PROGRAM MAIN
VAR
    //_tcoTestContext : TcoTestContext;
    _wpfContext : WpfContext;
    _wpfContextCall : BOOL := FALSE;
END_VAR

//_tcoIrc5TestContext.ProbeRun();
IF _wpfContextCall THEN
    _wpfContext.Run();
END_IF

END_PROGRAM

(* stored: Version 1.1.0.1, ProductVersion 3.1.4024.12
   POU MAIN: Id {d09427fb-b58f-0403-1aab-1726c3745601}, SpecialFunc None *)
